FUNCTION_BLOCK FB_Lineaireuitschuifpin IMPLEMENTS ITF_Lineaireuitschuifpin
VAR_INPUT
	// Sensoren van de cilinders of ze zijn uitgeschoven of ingeschoven
	Sensor_uitgeschoven : BOOL; // Terugmelding cilinder met pin is uitgeschoven
	Sensor_ingeschoven : BOOL; // Terugmelding cilinder met pin is ingeschoven
END_VAR

VAR_OUTPUT
	// Fysieke uitgangen aan de ventielen
	Uitschuiven_output : BOOL; 
	Inschuiven_output : BOOL;
END_VAR

VAR
	// Interne variabelen
	Uitschuiven_Intern : BOOL; 
	Inschuiven_Intern : BOOL; 
	
	Status_Intern : E_LineaireactuatoruitschuifpinnenStatus;
	Uitgeschoven_Intern : BOOL; 
	Ingeschoven_Intern : BOOL; 
	Error_Intern : BOOL;
	
	// Timer voor foutdetectie
	MotionTimeout : TON; 
END_VAR

PROPERTY Error : BOOL
GET
Error := Error_Intern;
END_GET
END_PROPERTY

PROPERTY Ingeschoven : BOOL
GET
Ingeschoven := Ingeschoven_Intern;
END_GET
END_PROPERTY

PROPERTY Inschuiven : BOOL
GET
Inschuiven := Inschuiven_Intern;
END_GET
SET
VAR
	Waarde : BOOL;
END_VAR
Inschuiven_Intern := Waarde;
END_SET
END_PROPERTY

PROPERTY Status : E_LineaireactuatoruitschuifpinnenStatus
GET
Status := Status_Intern;
END_GET
END_PROPERTY

PROPERTY Uitgeschoven : BOOL
GET
Uitgeschoven := Uitgeschoven_Intern;
END_GET
END_PROPERTY

PROPERTY Uitschuiven : BOOL
GET
Uitschuiven := Uitschuiven_Intern;
END_GET
SET
VAR
	Waarde : BOOL;
END_VAR
Uitschuiven_Intern := Waarde;
END_SET
END_PROPERTY

METHOD Update : BOOL
// Sensorstatus opslaan
Uitgeschoven_Intern := Sensor_uitgeschoven;
Ingeschoven_Intern := Sensor_ingeschoven; 

// Standaard outputs
Uitschuiven_output := FALSE; 
Inschuiven_output := FALSE; 

// Fout resetten
IF Error_Intern AND (NOT Uitschuiven_Intern) AND (Inschuiven_Intern) THEN
	Error_Intern := FALSE;
END_IF

// Status van de lineaire actuator met uitschuif pinnen
CASE Status_Intern OF 
	
	E_LineaireactuatoruitschuifpinnenStatus.Idle:
		IF Uitschuiven_Intern THEN
			Status_Intern := E_LineaireactuatoruitschuifpinnenStatus.Uitschuiven;
			MotionTimeout(IN := TRUE, PT := T#3S);
		ELSIF Inschuiven_Intern THEN
			Status_Intern := E_LineaireactuatoruitschuifpinnenStatus.Inschuiven;
			MotionTimeout(IN := TRUE, PT := T#3S);
		END_IF
	
	E_LineaireactuatoruitschuifpinnenStatus.Uitschuiven:
		Uitschuiven_output := TRUE; 
		
		IF Uitgeschoven_Intern THEN
			Status_Intern := E_LineaireactuatoruitschuifpinnenStatus.Uitgeschoven;
			MotionTimeout(IN := FALSE);
		ELSIF MotionTimeout.Q THEN
			Status_Intern := E_LineaireactuatoruitschuifpinnenStatus.Error;
			Error_Intern := TRUE;
		END_IF
	
	E_LineaireactuatoruitschuifpinnenStatus.Inschuiven:
		Inschuiven_output := TRUE;
		
		IF Ingeschoven_Intern THEN
			Status_Intern := E_LineaireactuatoruitschuifpinnenStatus.Ingeschoven;
			MotionTimeout(IN := FALSE);
		ELSIF MotionTimeout.Q THEN
			Status_Intern := E_LineaireactuatoruitschuifpinnenStatus.Error;
			Error_Intern := TRUE;
		END_IF
	
	E_LineaireactuatoruitschuifpinnenStatus.Uitgeschoven:
		IF Inschuiven_Intern THEN
			Status_Intern := E_LineaireactuatoruitschuifpinnenStatus.Inschuiven;
			MotionTimeout(IN := TRUE, PT := T#3S;
		END_IF
	
	E_LineaireactuatoruitschuifpinnenStatus.Ingeschoven:
		IF Uitschuiven_Intern THEN
			Status_Intern := E_LineaireactuatoruitschuifpinnenStatus.Uitschuiven;
			MotionTimeout(IN := TRUE, PT := T#3S;
		END_IF
	
	E_LineaireactuatoruitschuifpinnenStatus.Error:
		Uitschuiven_output := FALSE; 
		Inschuiven_output := FALSE; 
END_CASE
END_METHOD

END_FUNCTION_BLOCK

(* stored: Version 1.1.0.1
   POU FB_Lineaireuitschuifpin: Id {3aed7838-cf13-43b5-9856-d0a4446344f2}, SpecialFunc None
   Folder Methods: Id {7cf5dbe4-9c1e-408b-a58c-f63234e26ccb}
   Folder Properties: Id {00085976-954c-491a-8fd6-1ca882c7ca8c}
   Property Error: Id {16a90c64-643a-4e74-9cf5-86d5283335d0}
   Get Get: Id {7c6c457e-663c-4742-9d70-3cecf2b913fb}
   Property Ingeschoven: Id {30d240aa-63a5-4890-b548-93d3475ffc53}
   Get Get: Id {b5a2b890-1a04-41d4-bfb9-d70b18a765a3}
   Property Inschuiven: Id {3e4234c6-f9dd-4a07-a08b-d4b6d3b50fb2}
   Get Get: Id {ab11d67f-eb04-43c4-8cda-92608a7581a2}
   Set Set: Id {39cce0d0-08b3-4452-8188-fcfe43851e1c}
   Property Status: Id {cb8204f7-4950-4a8c-8934-597798037ced}
   Get Get: Id {69e69824-d7d1-4e68-9749-08fcefec1925}
   Property Uitgeschoven: Id {ff237dbd-da6e-4a70-9ad8-5de6085a01ab}
   Get Get: Id {25eb561d-228f-4445-918d-04bb84c202f8}
   Property Uitschuiven: Id {6f1245d3-703d-49e6-b5c3-fc9f7e845239}
   Get Get: Id {f7b9b1a6-5888-427a-afcf-65bb1aae2110}
   Set Set: Id {eb1e9f54-ed02-41e3-868e-c7b5bf4a6b17}
   Method Update: Id {2e73f703-d45a-4545-a444-69799cb78195} *)
